TYPE REQUEST :
STRUCT
	Header			:UINT;		// Must be 0x1234
	Command			:UINT;		// Value according to the command table
	Data			:UDINT;		// data according to the actual command
END_STRUCT
END_TYPE

(* stored: Version 1.1.0.1
   DUT REQUEST: Id {d5a70c30-6d79-4759-b0b9-8ede75cca0c7} *)
